(* IEC 61131-3 sources: lc3-vendor-sqlite/src, 8 files *)

(* ---- SQLite_Connect.iecst ---- *)
{ extern_c }
/*
 * Connects to a sqlite database.											 <br>
 * For more information about the SQLite connect:                            <br>
 * http://www.sqlite.org/c3ref/open.html							         <br>
 *                                                                           <br>
 * <b>dbname</b> = Path to the sqlite database file.					     <br>
 *
 * Returns the handle to the SQLite database.
 */
FUNCTION SQLite_Connect : lint

	VAR_INPUT
		dbname : String[100];
	END_VAR

	VAR_OUTPUT
		handle : lint;
	END_VAR

END_FUNCTION

(* ---- SQLite_Disconnect.iecst ---- *)
{ extern_c }
/*
 * Disconnects from a SQLite database.				    					 <br>
 * For more information about the SQLite disconnect:                         <br>
 * http://www.sqlite.org/c3ref/close.html							         <br>
 *                                                                           <br>
 * <b>handle</b> = Handle for the SQLite database opened by SQLite_Connect.  <br>
 *
 * Returns a value for troubleshooting.
 */
FUNCTION SQLite_Disconnect : int

	VAR_INPUT
		handle : lint;
	END_VAR

	VAR_OUTPUT
		response : int;
	END_VAR

END_FUNCTION

(* ---- SQLite_ExecuteStatement.iecst ---- *)
{ extern_c }
/*
 * Exectues a SQLite statement  .											 <br>
 * For more information about the SQLite execute:                            <br>
 * http://www.sqlite.org/c3ref/exec.html							         <br>
 *                                                                           <br>
 * <b>sql</b> = The SQL statement.										     <br>
 * <b>handle</b> = Handle for the SQLite database opened by SQLite_Connect.  <br>
 *
 * Returns a code for troubleshooting.
 */
FUNCTION SQLite_ExecuteStatement : int

	VAR_INPUT
		sql : String[500];
		handle : lint;
	END_VAR

	VAR_OUTPUT
		sqlresponse : int;
	END_VAR

END_FUNCTION

(* ---- SQLite_GetIntegers.iecst ---- *)
{ extern_c }
/*
 * Exectues a SQLite statement and returns the challanged values.			 <br>
 * For more information about the SQLite prepare & column_int:               <br>
 * http://www.sqlite.org/c3ref/prepare.html  						         <br>
 * http://www.sqlite.org/c3ref/column_blob.html                              <br>
 * 																			 <br>
 * <b>sql</b> = The SQL statement.										     <br>
 * <b>handle</b> = Handle for the SQLite database opened by SQLite_Connect.  <br>
 *
 * Returns an array of ints, filled as the select statement was written.
 */
FUNCTION SQLite_GetIntegers : ARRAY[0..9] of int

	VAR_INPUT
		handle : lint;
		sql : String[500];
	END_VAR

	VAR_OUTPUT
		integers : ARRAY[0..9] of int;
	END_VAR

END_FUNCTION

(* ---- SQLite_GetString.iecst ---- *)
{ extern_c }
/*
 * Exectues a SQLite statement and returns the challanged value.			 <br>
 * For more information about the SQLite prepare & column_text               <br>
 * http://www.sqlite.org/c3ref/prepare.html  						         <br>
 * http://www.sqlite.org/c3ref/column_blob.html                              <br>
 * 																			 <br>
 * <b>sql</b> = The SQL statement.										     <br>
 * <b>handle</b> = Handle for the SQLite database opened by SQLite_Connect.  <br>
 *
 * Returns a string of max. 50 chars, all above will be cut.
 */
FUNCTION SQLite_GetString : String[50]

	VAR_INPUT
		handle : lint;
		sql : String[500];
	END_VAR

	VAR_OUTPUT
		retstr : String[50];
	END_VAR

END_FUNCTION

(* ---- SQLite_GetTimestamp.iecst ---- *)
{ extern_c }
/*
 * Returns the current timestamp in unixepoch format.						 <br>
 * For more information about the bash time command:           			     <br>
 * http://ss64.com/bash/time.html				                             <br>
 * 																			 <br>
 * Returns an string of ten chars of the current timestamp in unixepoch.
 */
FUNCTION SQLite_GetTimestamp : STRING[10]

	VAR_OUTPUT
		timestamp : STRING[10];
	END_VAR

END_FUNCTION

(* ---- SQLite_StatementReplacer.iecst ---- *)
{ extern_c }
/*
 * Replaces the given string with the given variables.						 <br>
 * 																			 <br>
 * <b>string1</b> = The string where the variables should be replaced.	     <br>
 * <b>ints</b> = An array of ints which will be replaced in the string.	     <br>
 * <b>str</b> = A string which will be replaced in the string.				 <br>
 *
 * Returns a string of max. 500 chars with all the variables replaced.
 */
FUNCTION SQLite_StatementReplacer : STRING[500]
	VAR_INPUT
		string1 : string[400];
		ints : array[0..9] of int;
		str : string[50];
	END_VAR

	VAR_OUTPUT
		retstr : STRING[500];
	END_VAR

END_FUNCTION

(* ---- program.iecst ---- *)
/*
 * This is an example code for using the SQLite Vendor POUs in Logi.CAD3
 */
PROGRAM Template

	VAR
		str : STRING[100];
		handle : lint := 0;
		timestamp :STRING[10];
		sqlstring1: string[250];
		statement : STRING[500];
		ints : array[0..9] of int;

		sqlresponse : int;
		stri : string[50];
		integers : ARRAY[0..9] of int;

	END_VAR

		if handle = 0 then //opens the database handle if not already opened
		str := '/usr/local/DatabaseFiles/exampleDB';
		SQLite_Connect(dbname:=str,handle=>handle, ENO => ENO); end_if;

		//Getting the actual timestamp in unixepoch
		SQLite_GetTimestamp(timestamp => timestamp);

		//dummy value
		ints[0] := 5;

		//make an insert sql statement
		sqlstring1 :='insert into log("time", "value") values(}s, }0)';

 		//replace the variables with values
		SQLite_Sprintf(string1 := sqlstring1, str := timestamp, ints := ints, retstr => statement);

		//execute the sql statement
		SQLite_ExecuteStatement(handle := handle, sql := statement, sqlresponse => sqlresponse, ENO => ENO);

		//get the time of the last insert as formated string
		sqlstring1 :='select datetime(time, "unixepoch") from log where id like (select max("id") from log)';

		//execute the select statement and get the string
		SQLite_GetString(handle := handle, sql := sqlstring1, retstr => stri, ENO => ENO);

		//get the amount of rows in the log table
		sqlstring1 :='select count("id") from log';

		//execute and get the result as int
		SQLite_GetIntegers(handle := handle, sql := sqlstring1, integers => integers, ENO => ENO);

END_PROGRAM
